TYPE E_Mfr_NotifySeverity :
(
	eInfo		:= 0,
	eWarning	:= 1,
	eError		:= 2
);
END_TYPE

(* stored: Version 1.1.0.1
   DUT E_Mfr_NotifySeverity: Id {a3b5e7c1-d294-4f86-b1a2-8e4c9f3d7052} *)
